TYPE EL5101_Control :
STRUCT
	{attribute addProperty Name "Enable latch C"}
	EnableLatch_C : BIT;
	{attribute addProperty Name "Enable latch extern on positive edge"}
	EnableLatchExternOnPositiveEdge : BIT;
	{attribute addProperty Name "Set counter"}
	SetCounter : BIT;
	{attribute addProperty Name "Enable latch extern on negative edge"}
	EnableLatchExternOnNegativeEdge : BIT;
	{attribute 'hide'}
	{attribute addProperty Name "Bit 5(address x.4)"}
	Bit_5 : BIT;
	{attribute 'hide'}
	{attribute addProperty Name "Bit 6(address x.5)"}
	Bit_6 : BIT;
	{attribute 'hide'}
	{attribute addProperty Name "Bit 7(address x.6)"}
	Bit_7 : BIT;
	{attribute 'hide'}
	{attribute addProperty Name "Bit 8(address x.7)"}
	Bit_8 : BIT;
	{attribute 'hide'}
	{attribute addProperty Name "Bit 9(address x+1.0)"}
	Bit_9 : BIT;
	{attribute 'hide'}
	{attribute addProperty Name "Bit 10(address x+1.1)"}
	Bit_10 : BIT;
	{attribute 'hide'}
	{attribute addProperty Name "Bit 11(address x+1.2)"}
	Bit_11 : BIT;
	{attribute 'hide'}
	{attribute addProperty Name "Bit 12(address x+1.3)"}
	Bit_12 : BIT;
	{attribute 'hide'}
	{attribute addProperty Name "Bit 13(address x+1.4)"}
	Bit_13 : BIT;
	{attribute 'hide'}
	{attribute addProperty Name "Bit 14(address x+1.5)"}
	Bit_14 : BIT;
	{attribute 'hide'}
	{attribute addProperty Name "Bit 15(address x+1.6)"}
	Bit_15 : BIT;
	{attribute 'hide'}
	{attribute addProperty Name "Bit 16(address x+1.7)"}
	Bit_16 : BIT;
END_STRUCT
END_TYPE

(* stored: Version 1.1.0.1, ProductVersion 3.1.4024.9
   DUT EL5101_Control: Id {5d8c2ca7-7a2f-0d7c-024b-2cc49b33ead3} *)
